DATA_BLOCK "SPL"	// DB 18
TITLE = SPL dataarea
AUTHOR : NUMERIK
FAMILY : _800D
NAME : Basics
VERSION : 1.5
  STRUCT
   INSEP_VALID : ARRAY  [1 .. 8 ] OF BOOL ;	//used external SPL-Inputbytes(HW)
   OUTSEP_VALID : ARRAY  [1 .. 8 ] OF BOOL ;	//used external SPL-Outputbytes(HW)
   INSEP_ADDR : ARRAY  [1 .. 8 ] OF INT ;	//Addresses external SPL-Inputbytes(HW)
   OUTSEP_ADDR : ARRAY  [1 .. 8 ] OF INT ;	//Addresses external SPL-Outputbytes(HW)
   SPL_READY : BOOL ;	//setup finished
   STOP_MODE : BOOL ;	//0= Stop D, 1=Stop E
   SPL_DATA : STRUCT
    INSEP : ARRAY  [1 .. 64 ] OF BOOL ;
    OUTSEP : ARRAY  [1 .. 64 ] OF BOOL ;
    INSIP : ARRAY  [1 .. 64 ] OF BOOL ;
    OUTSIP : ARRAY  [1 .. 64 ] OF BOOL ;
    MARKERSIP : ARRAY  [1 .. 64 ] OF BOOL ;
   END_STRUCT ;
   SPL_DELTA : STRUCT 	//edge difference NCK - PLC for Diagnostic
    INSEP : ARRAY  [1 .. 64 ] OF BOOL ;
    OUTSEP : ARRAY  [1 .. 64 ] OF BOOL ;
    INSIP : ARRAY  [1 .. 64 ] OF BOOL ;
    OUTSIP : ARRAY  [1 .. 64 ] OF BOOL ;
    MARKERSIP : ARRAY  [1 .. 64 ] OF BOOL ;
   END_STRUCT ;
   CMDSI : BOOL ;	//multiplication of Timeout Value by Factor 10
   CMDSI_R1 : BOOL ;	//for future use
   CMDSI_R2 : BOOL ;	//for future use
   CMDSI_R3 : BOOL ;	//for future use
   CMDSI_R4 : BOOL ;	//for future use
   CMDSI_R5 : BOOL ;	//for future use
   CMDSI_R6 : BOOL ;	//for future use
   CMDSI_R7 : BOOL ;	//for future use
   STATUS_R0 : BOOL ;	//for future use
   STATUS_R1 : BOOL ;	//for future use
   STATUS_R2 : BOOL ;	//for future use
   STATUS_R3 : BOOL ;	//for future use
   STATUS_R4 : BOOL ;	//for future use
   COMM_TO : BOOL ;	//Communication Timeout
   STATUS_R6 : BOOL ;	//for future use
   STATUS_R7 : BOOL ;	//for future use
   STATSI : DINT ;	//Status: 0 - no error, 1 - 320 error number
   LEVELSI : DINT ;	//stacklevel SPL-KDV for Diagnostic
   PLCSIOUT : ARRAY  [1 .. 32 ] OF BOOL ;	//Single Channel Signals from NCK
   PLCSIIN : ARRAY  [1 .. 32 ] OF BOOL ;	//Single Channel Signals to NCK
   SPL_STATUS : ARRAY  [1 .. 16 ] OF BOOL ;	//SPL Status from NCK
   INSEP_PROFISAFE : ARRAY  [1 .. 8 ] OF BOOL ;	//external SPL-Inputbytes(HW) with PROFIsafe Slaves
   OUTSEP_PROFISAFE : ARRAY  [1 .. 8 ] OF BOOL ;	//external SPL-Outputbytes(HW) with PROFIsafe Slaves
   NoOfAxisPerBlock : ARRAY  [1 .. 8 ] OF BYTE ;	//Pointer and Tables for Teststop
   BlockPointer : ARRAY  [1 .. 8 ] OF BYTE ;
   AxisTable : ARRAY  [1 .. 31 ] OF BYTE ;
   FSDP : ARRAY  [1 .. 3 ] OF STRUCT
    ERR_REAC : INT ;	// IN: Error reaction
    ERROR : BOOL ;	// OUT: 1=Communication error
    SUBS_ON : BOOL ;	// OUT: 1=Receiver outputs fail-safe values
    DIAG : WORD ;	// OUT: Service information
    RETVAL14 : WORD ;	// OUT: Error code of SFC 14
    RETVAL15 : WORD ;	// OUT: Error code of SFC 15
   END_STRUCT ;
   FRDP : ARRAY  [1 .. 3 ] OF STRUCT
    SUBS : ARRAY  [0 .. 15 ] OF BOOL ;	// IN: Fail-safe value for receive data BOOL 00 ... BOOL 15
    ERR_REAC : INT ;	// IN: Error reaction
    ACK_REI : BOOL ;	// IN: 1=Acknowledgment for reintegration of send data following communication er
    RES1 : BOOL ;	//Reserved
    RES2 : BOOL ;	//Reserved
    RES3 : BOOL ;	//Reserved
    RES4 : BOOL ;	//Reserved
    RES5 : BOOL ;	//Reserved
    RES6 : BOOL ;	//Reserved
    RES7 : BOOL ;	//Reserved
    ERROR : BOOL ;	// OUT: 1=Communication error
    SUBS_ON : BOOL ;	// OUT: 1=Fail-safe values are output
    ACK_REQ : BOOL ;	// OUT: 1=Acknowledgment for reintegration of send data required
    SENDMODE : BOOL ;	// OUT: 1=F_CPU with F_SENDDP in deactivated safety mode
    DIAG : WORD ;	// OUT: Service information
    RETVAL14 : WORD ;	// OUT: Error code of SFC 14
    RETVAL15 : WORD ;	// OUT: Error code of SFC 15
   END_STRUCT ;
  END_STRUCT ;	
BEGIN
END_DATA_BLOCK

ORGANIZATION_BLOCK "OB 1"	// OB 1
VERSION : 1.0
VAR_TEMP
  OB1_EV_CLASS : BYTE ;
  OB1_SCAN_1 : BYTE ;
  OB1_PRIORITY : BYTE ;
  OB1_OB_NUMBR : BYTE ;
  OB1_RESERVED_1 : BYTE ;
  OB1_RESERVED_2 : BYTE ;
  OB1_PREV_CYCLE : INT ;
  OB1_MIN_CYCLE : INT ;
  OB1_MAX_CYCLE : INT ;
  OB1_DATE_TIME : DATE_AND_TIME ;
END_VAR
BEGIN
NETWORK
TITLE =
      CALL  "GP_HP";
//Insert User program from here
END_ORGANIZATION_BLOCK

ORGANIZATION_BLOCK OB 40
VERSION : 1.0
VAR_TEMP
  OB40_EV_CLASS : BYTE ;
  OB40_STRT_INF : BYTE ;
  OB40_PRIORITY : BYTE ;
  OB40_OB_NUMBR : BYTE ;
  OB40_RESERVED_1 : BYTE ;
  OB40_MDL_ID : BYTE ;
  OB40_MDL_ADDR : INT ;
  OB40_POINT_ADDR : DWORD ;
  OB40_DATE_TIME : DATE_AND_TIME ;	//data for the Basic program
  GP_IRFromNCK : BOOL ;	//Interrupt from NCK
  GP_TM : BOOL ;	//Toolmanagment
  GP_InPosition : ARRAY  [1 .. 31 ] OF BOOL ;	//InPos Signal from FC15,16,18
  GP_AuxFunction : ARRAY  [1 .. 10 ] OF BOOL ;	//auxiliary functions
  GP_FMBlock : ARRAY  [1 .. 10 ] OF BOOL ;	//not used
//Insert User-data from here
END_VAR
BEGIN
NETWORK
TITLE =
      CALL  "GP_PRAL";
//Insert User program from here
END_ORGANIZATION_BLOCK

ORGANIZATION_BLOCK OB 82
TITLE = "I/O Point Fault"
VERSION : 1.0
VAR_TEMP
  OB82_EV_CLASS : BYTE ;	//16#39, Event class 3, Entering event state, Internal fault event
  OB82_FLT_ID : BYTE ;	//16#XX, Fault identifcation code
  OB82_PRIORITY : BYTE ;	//Priority of OB Execution
  OB82_OB_NUMBR : BYTE ;	//82 (Organization block 82, OB82)
  OB82_RESERVED_1 : BYTE ;	//Reserved for system
  OB82_IO_FLAG : BYTE ;	//Input (01010100), Output (01010101)
  OB82_MDL_ADDR : WORD ;	//Base address of module with fault
  OB82_MDL_DEFECT : BOOL ;	//Module defective
  OB82_INT_FAULT : BOOL ;	//Internal fault
  OB82_EXT_FAULT : BOOL ;	//External fault
  OB82_PNT_INFO : BOOL ;	//Point information
  OB82_EXT_VOLTAGE : BOOL ;	//External voltage low
  OB82_FLD_CONNCTR : BOOL ;	//Field wiring connector missing
  OB82_NO_CONFIG : BOOL ;	//Module has no configuration data
  OB82_CONFIG_ERR : BOOL ;	//Module has configuration error
  OB82_MDL_TYPE : BYTE ;	//Type of module
  OB82_SUB_MDL_ERR : BOOL ;	//Sub-Module is missing or has error
  OB82_COMM_FAULT : BOOL ;	//Communication fault
  OB82_MDL_STOP : BOOL ;	//Module is stopped
  OB82_WTCH_DOG_FLT : BOOL ;	//Watch dog timer stopped module
  OB82_INT_PS_FLT : BOOL ;	//Internal power supply fault
  OB82_PRIM_BATT_FLT : BOOL ;	//Primary battery is in fault
  OB82_BCKUP_BATT_FLT : BOOL ;	//Backup battery is in fault
  OB82_RESERVED_2 : BOOL ;	//Reserved for system
  OB82_RACK_FLT : BOOL ;	//Rack fault, only for bus interface module
  OB82_PROC_FLT : BOOL ;	//Processor fault
  OB82_EPROM_FLT : BOOL ;	//EPROM fault
  OB82_RAM_FLT : BOOL ;	//RAM fault
  OB82_ADU_FLT : BOOL ;	//ADU fault
  OB82_FUSE_FLT : BOOL ;	//Fuse fault
  OB82_HW_INTR_FLT : BOOL ;	//Hardware interupt input in fault
  OB82_RESERVED_3 : BOOL ;	//Reserved for system
  OB82_DATE_TIME : DATE_AND_TIME ;	//Date and time OB82 started
END_VAR
BEGIN
NETWORK
TITLE = Detailed Diagnosis in OB82 (interrupt)
      CALL  "GP_DIAG" (
           $1                       := TRUE);
END_ORGANIZATION_BLOCK

ORGANIZATION_BLOCK OB 86
TITLE = "Loss Of Rack Fault"
VERSION : 1.0
VAR_TEMP
  OB86_EV_CLASS : BYTE ;	//16#38/39 Event class 3
  OB86_FLT_ID : BYTE ;	//16#C1/C4/C5, Fault identifcation code
  OB86_PRIORITY : BYTE ;	//Priority of OB Execution
  OB86_OB_NUMBR : BYTE ;	//86 (Organization block 86, OB86)
  OB86_RESERVED_1 : BYTE ;	//Reserved for system
  OB86_RESERVED_2 : BYTE ;	//Reserved for system
  OB86_MDL_ADDR : WORD ;	//Base address of IM module in rack with fault
  OB86_RACKS_FLTD : ARRAY  [0 .. 31 ] OF BOOL ;	//Racks in fault
  OB86_DATE_TIME : DATE_AND_TIME ;	//Date and time OB86 started
END_VAR
BEGIN
NETWORK
TITLE = Detailed Diagnosis in OB86 (interrupt)
      CALL  "GP_DIAG" (
           $1                       := TRUE);
END_ORGANIZATION_BLOCK

ORGANIZATION_BLOCK OB 100
VERSION : 1.0
VAR_TEMP
  OB100_EV_CLASS : BYTE ;
  OB100_STRTUP : BYTE ;
  OB100_PRIORITY : BYTE ;
  OB100_OB_NUMBR : BYTE ;
  OB100_RESERVED_1 : BYTE ;
  OB100_RESERVED_2 : BYTE ;
  OB100_STOP : WORD ;
  OB100_RESERVED_3 : WORD ;
  OB100_RESERVED_4 : WORD ;
  OB100_DATE_TIME : DATE_AND_TIME ;
END_VAR
BEGIN
NETWORK
TITLE =
      CALL  "RUN_UP" , "gp_par" (
           DIW 0                    := 1,
           DIW 2                    := 0,
           DID 4                    := P#I 0.0,
           DIW 8                    := 0,
           DID 10                   := P#Q 0.0,
           DIW 14                   := 0,
           DID 16                   := P#Q 8.0,
           DIW 20                   := 0,
           DID 22                   := P#Q 12.0,
           DIW 26                   := 6);
//Insert User program from here
END_ORGANIZATION_BLOCK
